Fanuc KAREL source: kt00728.KL

-- PROVISIONAL review KL for V1013-1; original PC SHA256 ad090a9ca707c2c87979bc2ee2ca3382e7a556482ffd8df8bfd67072b282326a
-- Incomplete behavior may be omitted. Consult companion uncertainty JSON. Do not deploy.
PROGRAM KT00728
%NOLOCKGROUP
VAR
  OUT : BOOLEAN
-- UNRESOLVED_DECL C1 type=00001c
-- UNRESOLVED_DECL C2 type=00001c
BEGIN
  -- UNRESOLVED_PC offsets 5-15; opcodes 9D,22,A5
  -- UNRESOLVED_PC offsets 20-30; opcodes 9C,22,A5
  -- UNRESOLVED_PC offsets 35-45; opcodes 9D,22,A5
  -- UNRESOLVED_PC offsets 50-60; opcodes 9C,22,A5
  -- UNRESOLVED_PC offsets 65-80; opcodes 22,63,23
  -- UNRESOLVED_PC offsets 85-89; opcodes 7F
END KT00728
